// TIA Portal V17 export
// export: Created 2024-09-02T12:49:58.8439794Z, ExportSetting WithDefaults, DisplayName Totally Integrated Automation Portal, DisplayVersion V17, DisplayName TIA Portal Openness, DisplayVersion V17, DisplayName TIA Portal Version Control Interface, DisplayVersion V17, DisplayName STEP 7 Professional, DisplayVersion V17, DisplayName STEP 7 Safety, DisplayVersion V17, DisplayName WinCC Professional, DisplayVersion V17
ORGANIZATION_BLOCK "LTLL_HMILite"   // OB550, LAD, ProgramCycle
TITLE = LTLL_HMILite / "Main Program Sweep (Cycle)"
{ S7_Optimized_Access := 'TRUE' }
AUTHOR : Siemens
FAMILY : HMI_Lite
NAME : LTLL_HMILite
VERSION : 8.10
// stored: AutoNumber true, IsIECCheckEnabled false, SetENOAutomatically false
   VAR_INPUT
      Initial_Call : Bool;   // Initial call of this OB
      Remanence : Bool;   // =True, if remanent data are available
   END_VAR
BEGIN

REGION Network 1: Calling up the HMI Lite functions for the first HMI / Aufruf der HMI Lite Funktionen für erstes HMI
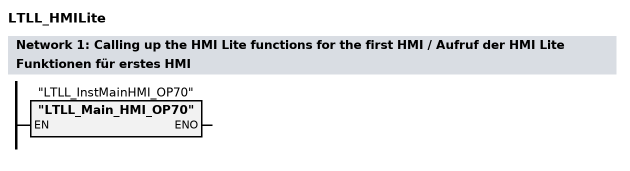
   RUNG wire#powerrail
      "LTLL_InstMainHMI_OP70"()
   END_RUNG
   // the same network as SCL:
   "LTLL_InstMainHMI_OP70"();   // "LTLL_Main_HMI_OP70"
END_REGION
END_ORGANIZATION_BLOCK
